(* PLC project Unnamed, Unknown Unnamed 1 *)
(* stored: creationDateTime 2025-06-20T20:22:35, modificationDateTime 2025-06-20T21:11:18 *)

PROGRAM assign
  VAR
    input1 AT %IX100.0 : BOOL := TRUE;
    input2 AT %IX100.1 : BOOL := FALSE;
    output1 AT %QX100.0 : BOOL;
    output2 AT %QX100.1 : BOOL;
  END_VAR

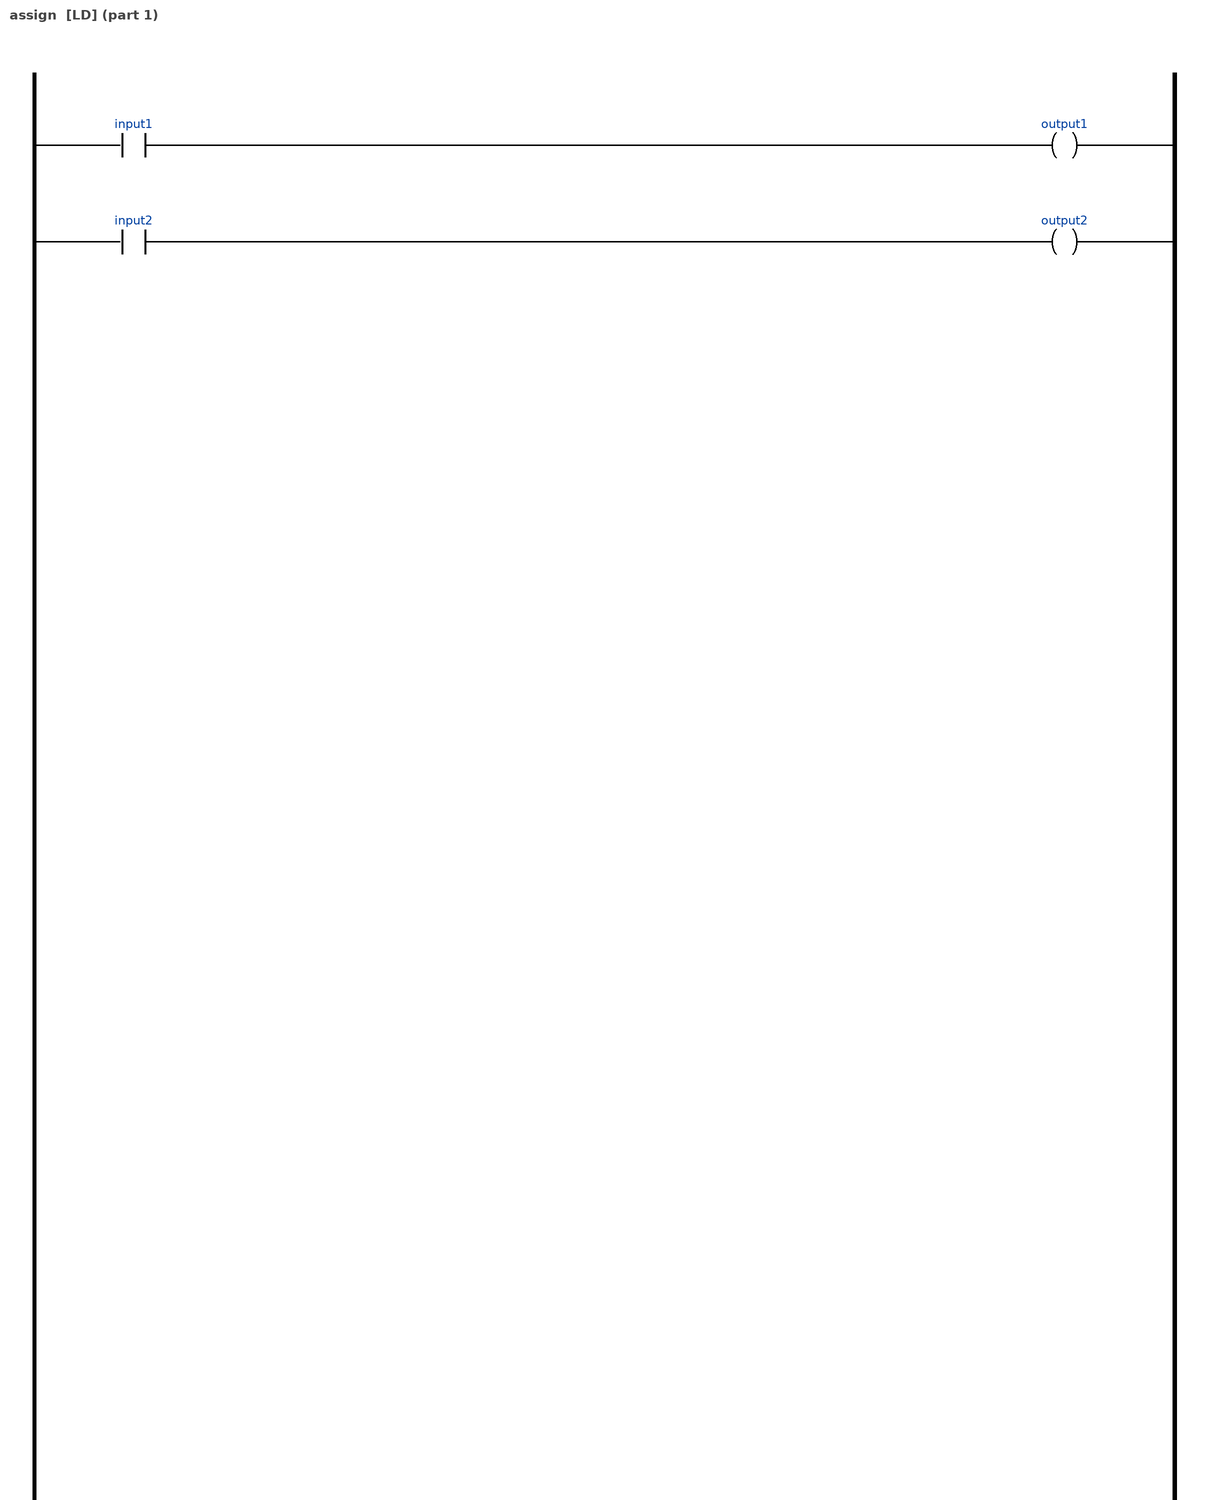
(* LD diagram, written out as Structured Text *)
output1 := input1;
output2 := input2;
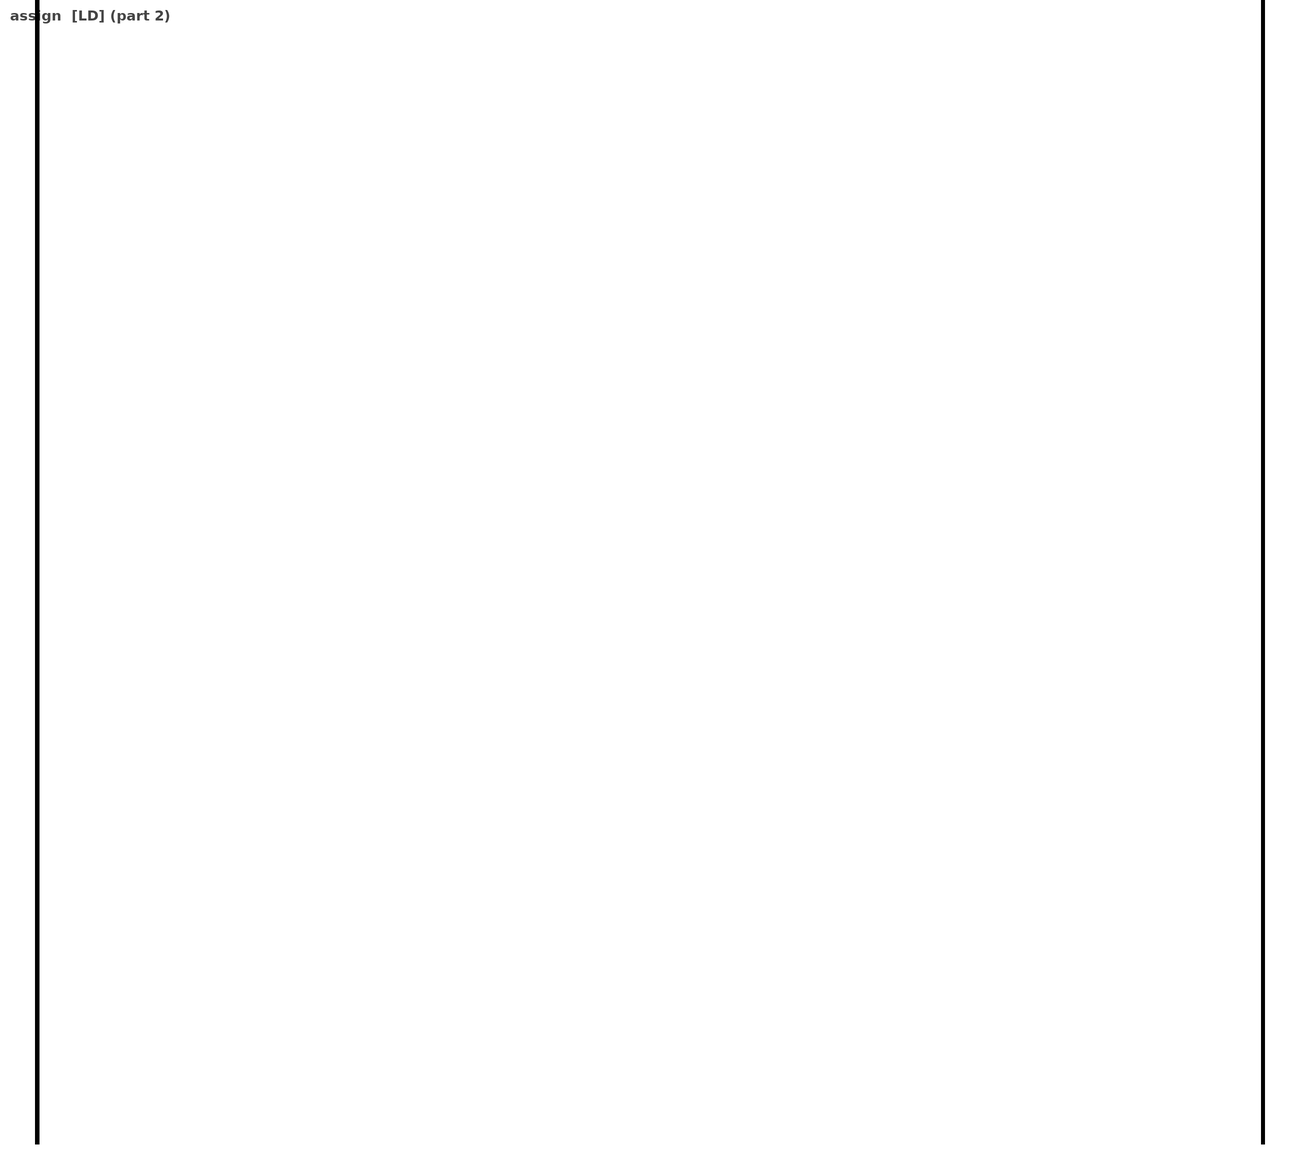
END_PROGRAM

CONFIGURATION Config0
  RESOURCE Res0 ON PLC
    TASK task0(INTERVAL := T#20ms, PRIORITY := 0);
    PROGRAM instance0 WITH task0 : assign;
  END_RESOURCE
END_CONFIGURATION
